// TIA Portal V19 export
TYPE "WkClockSet"
// stored: Access Published
   STRUCT
      Set_ON : Time_Of_Day;
      Set_OFF : Time_Of_Day;
      Enable : Bool;
   END_STRUCT;
END_TYPE
